FUNCTION_BLOCK Q_ChangePolygonScale (* Command Change Polygon Scale( Part 6 - F.54 ) *)
  (* Standard: ISO 11783-6; Description: This command is used by a Working Set to change the scale of a complete Output Polygon object. Return values iso_s16 - E_NO_ERR - OK - E_OVERFLOW - buffer overflow - E_NOACT - Command not possible in current state - E_NO_INSTANCE - No VT client available *)
  (* Version 1.0, 2022-07-08, franz *)
  (* Documentation:
  This command is used by a Working Set to change the scale of a complete Output Polygon object.
   Return values
   iso_s16
    - E_NO_ERR - OK
   - E_OVERFLOW - buffer overflow
   - E_NOACT - Command not possible in current state
   - E_NO_INSTANCE - No VT client available
  *)
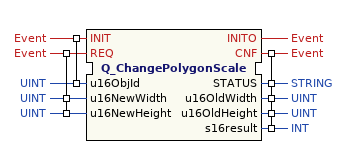
  EVENT_INPUT
    INIT WITH u16ObjId; (* Service Initialization *)
    REQ WITH u16NewWidth, u16NewHeight; (* Service Request *)
  END_EVENT
  EVENT_OUTPUT
    INITO; (* Initialization Confirm *)
    CNF WITH STATUS, s16result, u16OldWidth, u16OldHeight; (* Confirmation of Requested Service *)
  END_EVENT
  VAR_INPUT
    u16ObjId : UINT; (* Object ID of the Output Polygon object to change *)
    u16NewWidth : UINT; (* New width attribute *)
    u16NewHeight : UINT; (* New height attribute *)
  END_VAR
  VAR_OUTPUT
    STATUS : STRING; (* Service Status *)
    u16OldWidth : UINT; (* Old width attribute *)
    u16OldHeight : UINT; (* Old height attribute *)
    s16result : INT; (* retval see description *)
  END_VAR
END_FUNCTION_BLOCK
